(* CoDeSys 2.3 export: ERR_SET.EXP *)

(* POU Alarm/ERR_SET, ST *)
FUNCTION ERR_SET : BOOL
VAR_INPUT
	Num: INT; (* Номер ошибки *)
	Val: BOOL;(* Значение ошибки *)
END_VAR
VAR
END_VAR
	glbErrors[Num].State := Val;

	(* Если произошла ошибка и нужна регистрация, регистрируем ошибку *)

	IF Val AND NOT glbErrors[Num].StateM AND glbErrors[Num].Latch THEN
		glbErrors[Num].LatchState := TRUE;
	END_IF;

	glbErrors[Num].StateM := Val;
END_FUNCTION
